PROGRAM modbee
VAR
	MODBEE_HW_CONFIG0 : MODBEE_HW_CONFIG;
	MODBEE_CONFIG0 : MODBEE_CONFIG;
END_VAR

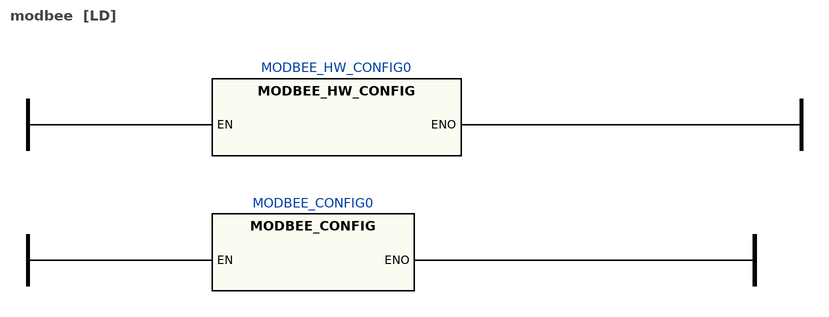
(* LD diagram, written out as Structured Text *)
MODBEE_HW_CONFIG0();
MODBEE_CONFIG0();
END_PROGRAM
